PROGRAM MAIN
VAR
END_VAR

END_PROGRAM

(* stored: Version 1.1.0.1
   POU MAIN: Id {d3a9a008-7083-4b93-8cc3-a19958ab080b} *)
